{attribute addProperty BoxType "EL3773-0000-0016"}
{attribute addProperty Id "U2_STATUSAT %I*U2_STATUS_F9B4A013162"}
{attribute addProperty CRC "274067627"}
{attribute addProperty SizeInBites "16"}
{attribute addProperty SizeInBytes "2"}
TYPE L2_Voltage_Status_1055F0AB :
STRUCT
	{attribute addProperty Name "U2_STATUS"}
	U2_STATUS AT %I* : U2_STATUS_F9B4A013;
END_STRUCT
END_TYPE

(* stored: Version 1.2.0.0, ProductVersion 3.1.4024.9
   DUT L2_Voltage_Status_1055F0AB: Id {154ecb0b-fcaf-4998-9750-b72405c38a67} *)
